{attribute 'pack_mode' := '1'}  // needed for python pyads reading
TYPE ST_PartTrackingData :
STRUCT
	OK_ToProcess: BOOL;
	NOK_ToProcess: BOOL;
	bInitRun: BOOL;
	WellplateStatus: INT;
	WellplateNOK_Reason: INT;
	nDestinationProcess: UINT;
	nPriority: UINT;
	nSerial: UDINT;
	PuncherProcessResults: ARRAY[1..96] OF ST_ProcessResult;
	PipeteProcesResults: ARRAY[1..96] OF ST_ProcessResult;
	DoseProcesResult: ARRAY[1..12] OF ST_ProcessResult;
END_STRUCT
END_TYPE

(* stored: Version 1.1.0.1
   DUT ST_PartTrackingData: Id {7e2a9c1d-4f6b-4a3e-9d2c-1b8f5e6a0c37} *)
